// TIA Portal V17 export
// export: Created 2026-04-13T11:12:41.5072655Z, ExportSetting WithDefaults, DisplayName Totally Integrated Automation Portal, DisplayVersion V17 Update 4, DisplayName TIA Portal Openness, DisplayVersion V17 Update 4, DisplayName TIA Portal Version Control Interface, DisplayVersion V17, DisplayName SINAMICS Startdrive Advanced, DisplayVersion V17, DisplayName SINAMICS Startdrive G130, G150, S120, S150, SINAMICS MV, S210, DisplayVersion V17, DisplayName SINAMICS Startdrive G110M, G120, G120C, G120D, G120P, G115D, DisplayVersion V17, DisplayName STEP 7 Professional, DisplayVersion V17 Update 4, DisplayName STEP 7 Safety, DisplayVersion V17, DisplayName WinCC Professional, DisplayVersion V17 Update 4
FUNCTION_BLOCK "A4--电机控制"   // FB6, SCL
{ S7_Optimized_Access := 'TRUE' }
VERSION : 0.1
// stored: AutoNumber true, IsIECCheckEnabled false, IsRetainMemResEnabled false, MemoryReserve 100, SetENOAutomatically false, UDAEnableTagReadback false
   VAR_INPUT
      HMI上限 : Real := 50.0;
      HMI下限 : Real;
      PLC上限 : Int := 27648;
      PLC下限 : Int := 0;
      电机报警信号 : Bool;
      电机输入模拟量 : Int;
      电机输出最小 : Real;
   END_VAR
   VAR_OUTPUT
      电机输出反馈 : Real;
      电机报警输出 : Bool;
   END_VAR
   VAR_IN_OUT
      按钮_消警按钮 : Bool;
      模式设定 : Real;
      电机控制按钮 : Bool;
      频率设定 : Real;
      电机输出Q : Bool;
      电机速度AO : Int;
      动画 : Int;
      安全停机 : Bool;
   END_VAR
   VAR
      P1 : Bool;
      TON1 : TON_TIME;
      Temp_1 { S7_SetPoint := 'True'} : Int;
      DBD1 : Real;
      DBD2 : Real;
      DBD3 : Real;
   END_VAR
BEGIN

   //手动控制--------------------------------------------------------------------------------------------------------------
   IF #模式设定 = 2.0 OR #模式设定 = 3.0  OR #模式设定 = 4.0 OR #模式设定 = 5.0  THEN
       //预热器加热手动控制
       IF #电机控制按钮 THEN
           #电机输出Q := TRUE;
           (* #电机速度AO := REAL_TO_INT(#频率设定 * 27648.0 / 50.0); *)
           #DBD1 := NORM_X_REAL(MIN := #HMI下限, VALUE := #频率设定, MAX := #HMI上限);
           #电机速度AO := SCALE_X_INT(MIN := #PLC下限, VALUE := #DBD1, MAX := #PLC上限);
       ELSE
           #电机输出Q := FALSE;
       END_IF;
   END_IF;


   // 自动启动--------------------------------------------------------------------------------------------------------------
   IF #电机输出Q THEN
       (* #电机速度AO := REAL_TO_INT(#频率设定 * 27648.0 / 50.0); *)
       #DBD2 := NORM_X_REAL(MIN := #HMI下限, VALUE := #频率设定, MAX := #HMI上限);
       #电机速度AO := SCALE_X_INT(MIN := #PLC下限, VALUE := #DBD2, MAX := #PLC上限);
   END_IF;
   IF NOT #电机输出Q THEN
       #电机速度AO := 0;
   END_IF;

   IF #电机报警输出 THEN
       #电机速度AO := 0;
       #电机控制按钮 := FALSE;
       #电机输出Q := FALSE;
   END_IF;


   IF #电机输出Q THEN
       #DBD3 := NORM_X_REAL(MIN := #PLC下限, VALUE := #电机输入模拟量, MAX := #PLC上限);
       #电机输出反馈 := SCALE_X_REAL(MIN := #HMI下限, VALUE := #DBD3, MAX := #HMI上限);
   ELSE
       #电机输出反馈 := 0;
   END_IF;
   #TON1(IN := #电机输出Q AND #电机输出反馈  < #电机输出最小,
                          PT := T#60s,
                          Q => #P1);

   IF #P1 OR #电机报警信号 THEN
       #电机报警输出 := TRUE;
   ELSE
       #电机报警输出 := FALSE;
   END_IF; 

   IF
       #模式设定 = 1 AND #电机报警输出 THEN

       #安全停机 := 1;
   END_IF;

   IF #按钮_消警按钮 THEN
       #P1 := FALSE;
       #电机报警输出 := FALSE;
   END_IF;

   IF #电机输出Q AND #频率设定 > #电机输出最小 THEN
       IF "Clock_10Hz" THEN
           #Temp_1 := #Temp_1 + 1;
       END_IF;

       IF #Temp_1 = 2 THEN
           #Temp_1 := 0;
       END_IF;
       IF #Temp_1 = 0 THEN
           #动画 := 0;
       END_IF;
       IF #Temp_1 = 1 THEN
           #动画 := 1;
       END_IF;

   END_IF;
   IF NOT #电机输出Q THEN
       #动画 := 0;
   END_IF;
END_FUNCTION_BLOCK
